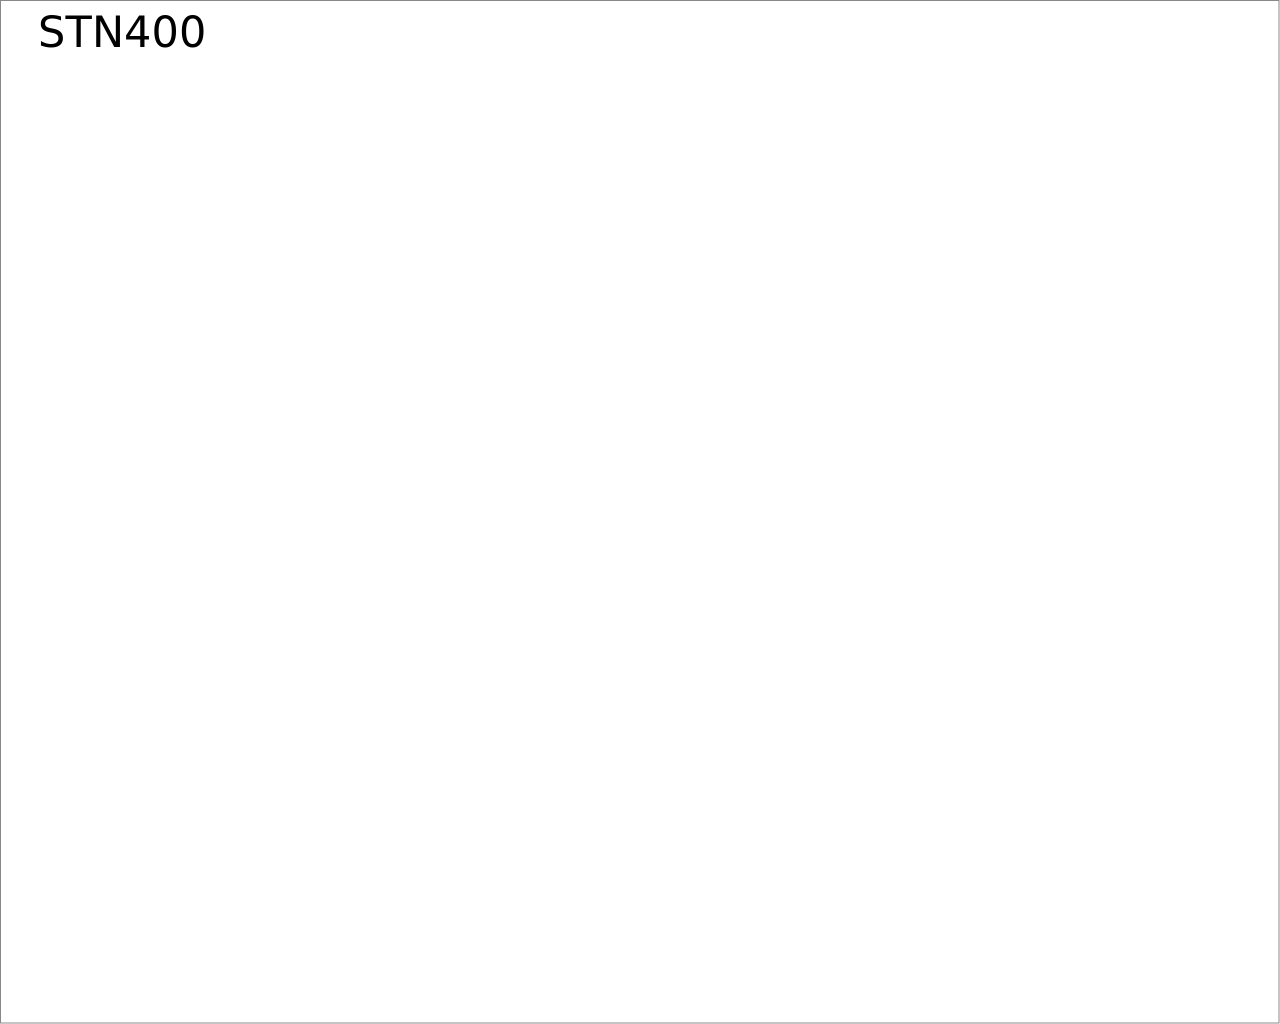
VISUALIZATION Visualization  // 1280x1024
    Label (3,0 239x64), "STN400"
END_VISUALIZATION

(* stored: Version 1.1.0.1, ProductVersion 3.1.4024.2
   Visu Visualization: Id {1ca4161e-ae0f-479c-9e89-d307cf9521bf} *)
